ABB RAPID module: TCP_tool2E2e.MOD

MODULE TCP_tool2E2e
	! Points are read in order of declaration.
  ! Please do not change the order of points!

  LOCAL PERS robtarget pTCP_Point1:=[[593.7265,7.185209,326.2721],[0.418707460165024,-0.00928415916860104,0.907616913318634,0.0287987273186445],[0,1,-2,0],[9E+09,9E+09,9E+09,9E+09,9E+09,9E+09]];
	LOCAL PERS robtarget pTCP_Point2:=[[622.7628,-9.358312,324.8137],[0.000707637693267316,-0.938009023666382,-0.0704698711633682,0.33937081694603],[-1,1,-1,1],[9E+09,9E+09,9E+09,9E+09,9E+09,9E+09]];
	LOCAL PERS robtarget pTCP_Point3:=[[603.7779,-23.56993,324.0442],[0.374255806207657,-0.378982186317444,0.820272147655487,0.208467274904251],[-1,0,-2,0],[9E+09,9E+09,9E+09,9E+09,9E+09,9E+09]];
	LOCAL PERS robtarget pTCP_Point4:=[[608.5183,24.88917,326.4019],[0.340109407901764,0.562201261520386,0.730407774448395,-0.186439588665962],[0,-1,1,0],[9E+09,9E+09,9E+09,9E+09,9E+09,9E+09]];

ENDMODULE
